FUNCTION_BLOCK DebugList
VAR
	_refDebug			: REFERENCE TO ARRAY[0..Param.nMaxDebugArraySize] OF ST_DebugInfo REF= _Debug.stDebug;
END_VAR

END_FUNCTION_BLOCK

(* stored: Version 1.1.0.1
   POU DebugList: Id {988c50c4-c1a3-41fc-bd18-6efe33b318e2}, SpecialFunc None *)
